TYPE TileInfoType :
STRUCT
	Center 	: LREAL;
	East 	: LREAL;
	North 	: LREAL;
	South	: LREAL;
	West 	: LREAL;
	FanRPM	: UINT;
END_STRUCT
END_TYPE

(* stored: Version 1.1.0.1, ProductVersion 3.1.4024.12
   DUT TileInfoType: Id {f645aefc-2d00-4022-8576-97566943d0dc} *)
